// TIA Portal V17 export
// export: Created 2025-06-26T07:49:52.416455Z, ExportSetting WithDefaults, DisplayName Totally Integrated Automation Portal, DisplayVersion V17 Update 8, DisplayName TIA Portal Openness, DisplayVersion V17 Update 8, DisplayName TIA Portal Version Control Interface, DisplayVersion V17, DisplayName STEP 7 Professional, DisplayVersion V17 Update 8, DisplayName STEP 7 Safety, DisplayVersion V17 Update 6, DisplayName WinCC Advanced, DisplayVersion V17 Update 8
VAR_GLOBAL   // PLC tag table "Inverters"
   TA1_Rx AT %I10.0 : "stABB_ACSx80_Rx";   // HBL-SC-01   {ExternalAccessible false, ExternalVisible false, ExternalWritable false}
   TA1_Tx AT %Q10.0 : "stABB_ACSx80_Tx";   // HBL-SC-01   {ExternalAccessible false, ExternalVisible false, ExternalWritable false}
   TA2_Rx AT %I30.0 : "stABB_ACSx80_Rx";   // HBL-SC-02   {ExternalAccessible false, ExternalVisible false, ExternalWritable false}
   TA10_Rx AT %I68.0 : "stABB_ACSx80_Rx";   // HBL-SC-10   {ExternalAccessible false, ExternalVisible false, ExternalWritable false}
   TA2_Tx AT %Q30.0 : "stABB_ACSx80_Tx";   // HBL-SC-02   {ExternalAccessible false, ExternalVisible false, ExternalWritable false}
   TA10_Tx AT %Q68.0 : "stABB_ACSx80_Tx";   // '   {ExternalAccessible false, ExternalVisible false, ExternalWritable false}
   TA_State AT %IB7 : Byte;   // 1 = online   {ExternalAccessible false, ExternalVisible false, ExternalWritable false}
   TA3_Rx AT %I228.0 : "stABB_ACSx80_Rx";   // HBL-SC-03   {ExternalAccessible false, ExternalVisible false, ExternalWritable false}
   TA3_Tx AT %Q88.0 : "stABB_ACSx80_Tx";   // HBL-SC-03   {ExternalAccessible false, ExternalVisible false, ExternalWritable false}
END_VAR
